(* Logix 5000 project; controller DIMTER vendor 1 type 14 code 77 rev 15.4; software revision 15.01; part 4 of 4 *)
(* tags used below, declared in another part *)
   BufferReady : TIMER;
   CurrentShift : DINT;   // Shift Currently Operating
   F : BOOL[2016];   // Flags
   FLASHER : TIMER;   // Lamp Flasher
   Oneshots : BOOL[128];
   RecordFault : BOOL;
   RecordPieceSaw1 : BOOL;   // Record Piece Count For Shift Total
   RecordPieceSaw2 : BOOL;   // Record Piece Count For Shift Total
   Saw1FailureDelay : TIMER;
   Saw2FailureDelay : TIMER;
   T : TIMER[100];   // Timers
   A120 : ALIAS FOR Local:4:O.Data.0;   // O:4.0/0 A12.0 Buffer Selection1
   A121 : ALIAS FOR Local:4:O.Data.1;   // O:4.0/1 A12/1 Buffer Selection 2
   A122 : ALIAS FOR Local:4:O.Data.2;   // O:4.0/2 A12.2 Reset Failure
   A130 : ALIAS FOR Local:4:O.Data.8;   // O:4.0/8 A13.0 Failure Conveyor
   A131 : ALIAS FOR Local:4:O.Data.9;   // O:4.0/9 A13.1 Failure Saw 1
   A132 : ALIAS FOR Local:4:O.Data.10;   // O:4.0/10 A13.2 Failure Saw 2
   A133 : ALIAS FOR Local:4:O.Data.11;   // O:4.0/11 A13.3 Defect Measuring Computer
   A134 : ALIAS FOR Local:4:O.Data.12;   // O:4.0/12 A13.4 Safety Barrier Transfer Station
   A137 : ALIAS FOR Local:4:O.Data.15;   // O:4.0/15 A137 Safety Barrier Transfer Station
   Delay : TIMER[30];   // Delay Timers
   E00 : ALIAS FOR Local:1:I.Data.0;   // I:1.0/0 E0.0 Control Power On
   E01 : ALIAS FOR Local:1:I.Data.1;   // I:1.0/1 E0.1 Saw Hood 1 Closed
   E02 : ALIAS FOR Local:1:I.Data.2;   // I:1.0/2 E0.2 Saw Motor 1 On
   E03 : ALIAS FOR Local:1:I.Data.3;   // I:1.0/3 E0.3 Release - Feed Saw 1
   E04 : ALIAS FOR Local:1:I.Data.4;   // I:1.0/4 E0.4 Failure Saw 1
   E05 : ALIAS FOR Local:1:I.Data.5;   // I:1.0/5 E0.5 Failure Chain Ejector
   E06 : ALIAS FOR Local:1:I.Data.6;   // I:1.0/6 E0.6 Failure Conveyor in Front of Saw 1
   E07 : ALIAS FOR Local:1:I.Data.7;   // I:1.0/7 E0.7 Failure Conveyor in Front of Saw 2
   E10 : ALIAS FOR Local:1:I.Data.8;   // I:1.0/8 E1.0 Failure Weinig Conveyor
   E106 : ALIAS FOR Local:3:I.Data.22;   // I:3.1/6 E10.6 Cross Belt 1 Cyclewise Continuous Running
   E11 : ALIAS FOR Local:1:I.Data.9;   // I:1.0/9 E1.1 Saw Hood 2 Closed
   E111 : ALIAS FOR Local:3:I.Data.25;   // I:3.1/9 E11.1 Cross Belt 2 Cyclewise Continuous Running
   E12 : ALIAS FOR Local:1:I.Data.10;   // I:1.0/10 E1.2 Saw Motor 2 On
   E13 : ALIAS FOR Local:1:I.Data.11;   // I:1.0/11 E1.3 Release - Feed Saw 2
   E14 : ALIAS FOR Local:1:I.Data.12;   // I:1.0/12 E1.4 Failure Saw 2
   E15 : ALIAS FOR Local:1:I.Data.13;   // I:1.0/13 E1.5 Data Ready At Saw
   E17 : ALIAS FOR Local:1:I.Data.15;   // I:1.0/15 E1.7 Defect Measuring Computer
   E20 : ALIAS FOR Local:1:I.Data.16;   // I:1.1/0 E2.0 Protection Hood Measuring System
   E22 : ALIAS FOR Local:1:I.Data.18;   // I:1.1/2 E2.2 Frequency Converter Rollcase in Front of Saw 1 Ready For Operation
   E23 : ALIAS FOR Local:1:I.Data.19;   // I:1.1/3 E2.3 Frequency Converter Rollcase in Front of Saw 2 Ready For Operation
   E24 : ALIAS FOR Local:1:I.Data.20;   // I:1.1/4 E2.4 Emergency Shutdown Internal
   E26 : ALIAS FOR Local:1:I.Data.22;   // I:1.1/6 E2.6 Safety Barrier at Transfer Station Closed
   E27 : ALIAS FOR Local:1:I.Data.23;   // I:1.1/7 E2.7 Reset Safety Barrier at Transfer Station
   E33 : ALIAS FOR Local:1:I.Data.27;   // I:1/1/11 E3.3 PE Behind Measurement Station
   E43 : ALIAS FOR Local:2:I.Data.3;   // I:2.0/3 E4.3 Infeed Saw 1 On
   E44 : ALIAS FOR Local:2:I.Data.4;   // I:2.0/4 E4.4 Waste Conveyor Belt On
   E47 : ALIAS FOR Local:2:I.Data.7;   // I:2.0/7 E4.7 Lamp Test
   E53 : ALIAS FOR Local:2:I.Data.11;   // I:2.0/11 E5.3 Infeed Saw 2 On
   E54 : ALIAS FOR Local:2:I.Data.12;   // I:2.0/12 E5.4 Measuring Station On
   Faults : BOOL[224];   // Fault Array
   HMI_IntWords : INT[200];   // Integer Words to HMI
   IntsFromHMI : INT[100];   // Integers From HMI
   RealTimeClock : DINT[10];
   Status : BOOL[224];   // Status Array
(* MainProgram, continued *)

ROUTINE ShiftControl   (* ladder *)
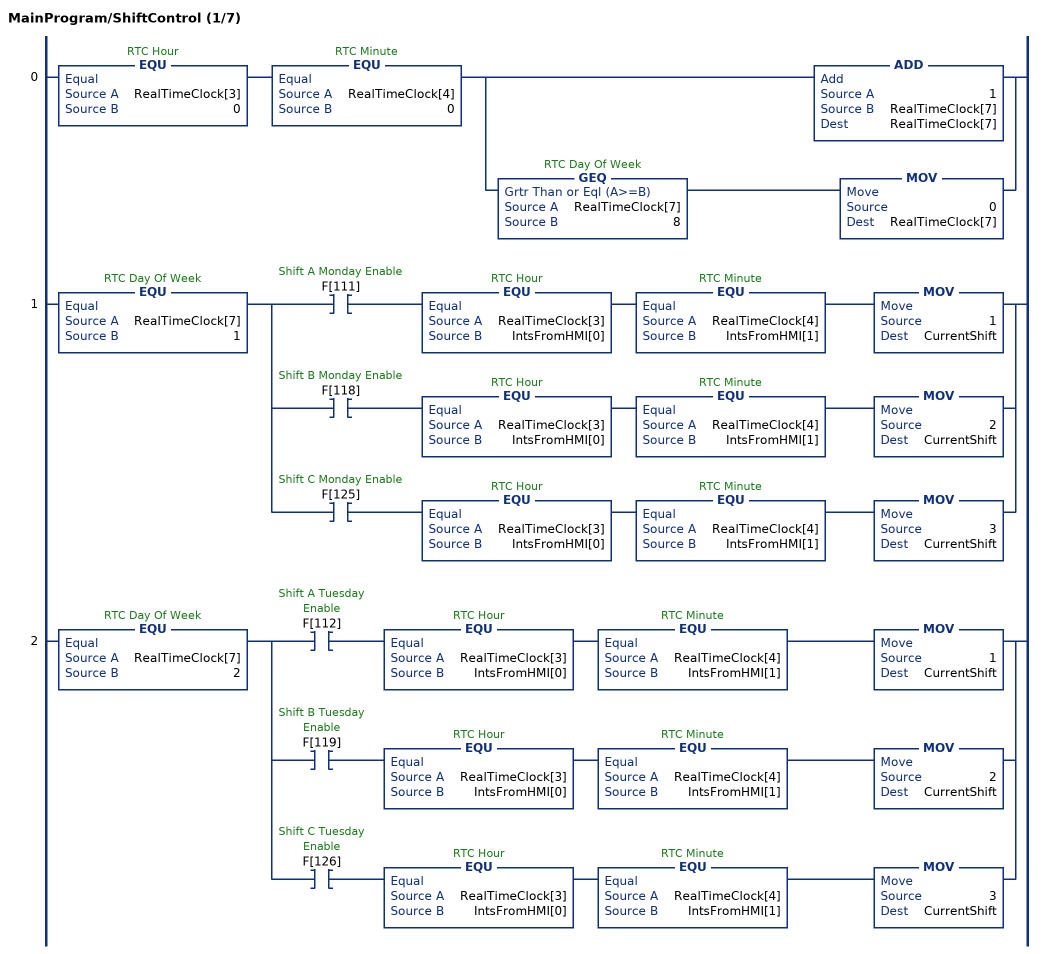
   0: EQU(RealTimeClock[3],0)EQU(RealTimeClock[4],0)[ADD(1,RealTimeClock[7],RealTimeClock[7]) ,GEQ(RealTimeClock[7],8) MOV(0,RealTimeClock[7]) ];
   1: EQU(RealTimeClock[7],1)[XIC(F[111]) EQU(RealTimeClock[3],IntsFromHMI[0]) EQU(RealTimeClock[4],IntsFromHMI[1]) MOV(1,CurrentShift) ,XIC(F[118]) EQU(RealTimeClock[3],IntsFromHMI[0]) EQU(RealTimeClock[4],IntsFromHMI[1]) MOV(2,CurrentShift) ,XIC(F[125]) EQU(RealTimeClock[3],IntsFromHMI[0]) EQU(RealTimeClock[4],IntsFromHMI[1]) MOV(3,CurrentShift) ];
   2: EQU(RealTimeClock[7],2)[XIC(F[112]) EQU(RealTimeClock[3],IntsFromHMI[0]) EQU(RealTimeClock[4],IntsFromHMI[1]) MOV(1,CurrentShift) ,XIC(F[119]) EQU(RealTimeClock[3],IntsFromHMI[0]) EQU(RealTimeClock[4],IntsFromHMI[1]) MOV(2,CurrentShift) ,XIC(F[126]) EQU(RealTimeClock[3],IntsFromHMI[0]) EQU(RealTimeClock[4],IntsFromHMI[1]) MOV(3,CurrentShift) ];
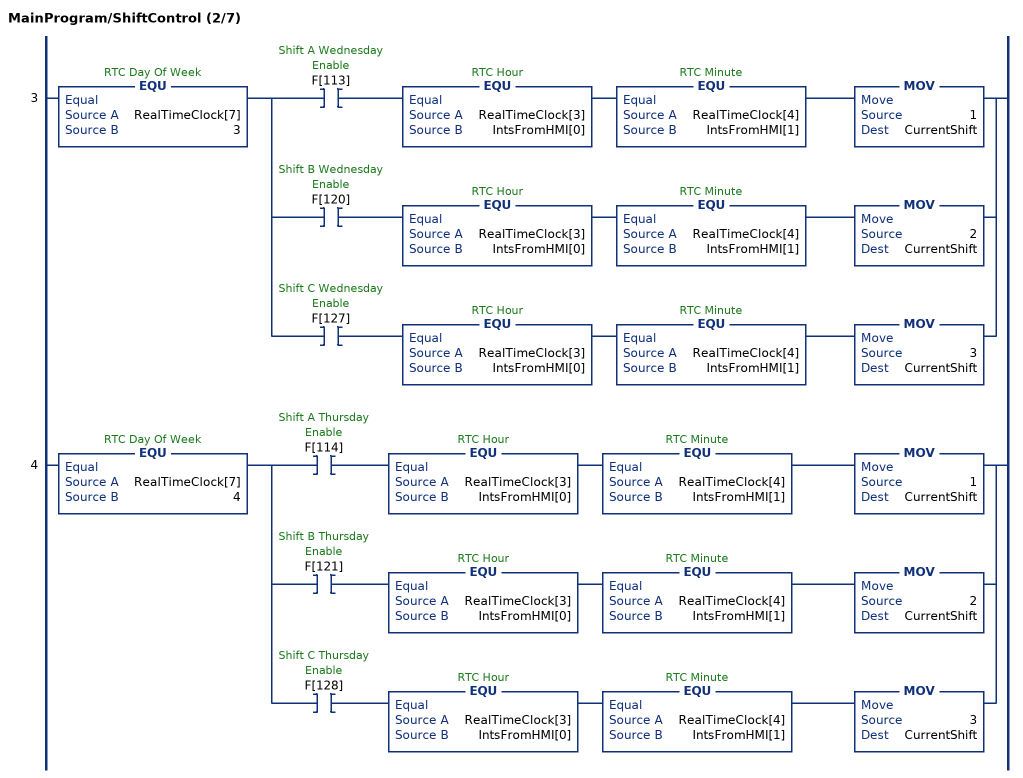
   3: EQU(RealTimeClock[7],3)[XIC(F[113]) EQU(RealTimeClock[3],IntsFromHMI[0]) EQU(RealTimeClock[4],IntsFromHMI[1]) MOV(1,CurrentShift) ,XIC(F[120]) EQU(RealTimeClock[3],IntsFromHMI[0]) EQU(RealTimeClock[4],IntsFromHMI[1]) MOV(2,CurrentShift) ,XIC(F[127]) EQU(RealTimeClock[3],IntsFromHMI[0]) EQU(RealTimeClock[4],IntsFromHMI[1]) MOV(3,CurrentShift) ];
   4: EQU(RealTimeClock[7],4)[XIC(F[114]) EQU(RealTimeClock[3],IntsFromHMI[0]) EQU(RealTimeClock[4],IntsFromHMI[1]) MOV(1,CurrentShift) ,XIC(F[121]) EQU(RealTimeClock[3],IntsFromHMI[0]) EQU(RealTimeClock[4],IntsFromHMI[1]) MOV(2,CurrentShift) ,XIC(F[128]) EQU(RealTimeClock[3],IntsFromHMI[0]) EQU(RealTimeClock[4],IntsFromHMI[1]) MOV(3,CurrentShift) ];
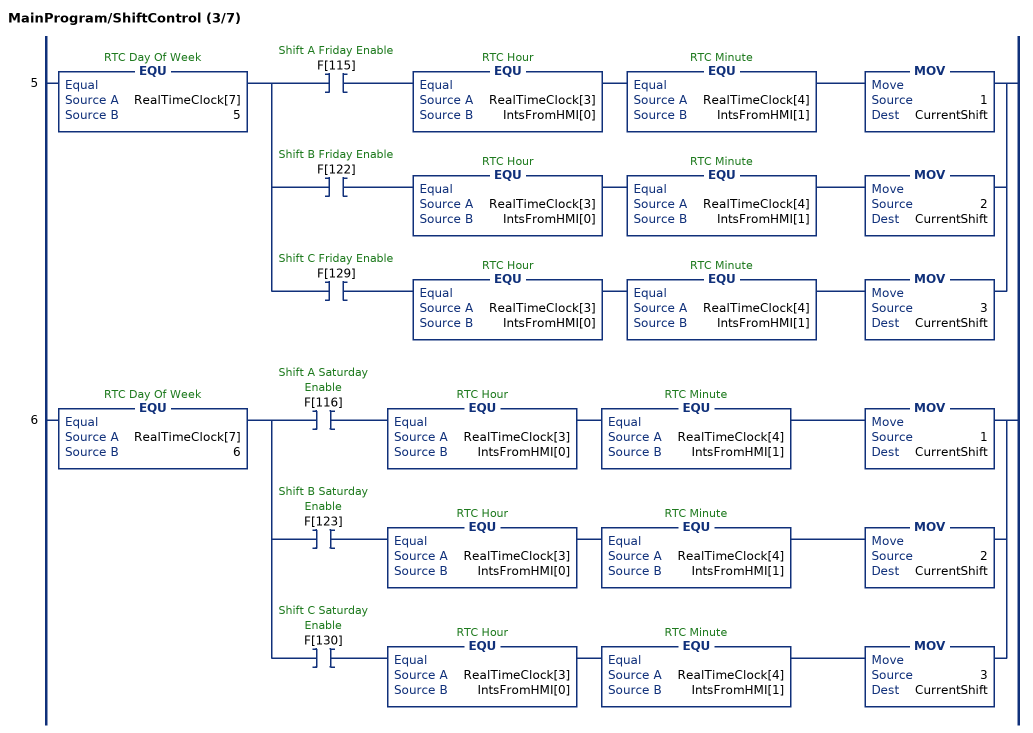
   5: EQU(RealTimeClock[7],5)[XIC(F[115]) EQU(RealTimeClock[3],IntsFromHMI[0]) EQU(RealTimeClock[4],IntsFromHMI[1]) MOV(1,CurrentShift) ,XIC(F[122]) EQU(RealTimeClock[3],IntsFromHMI[0]) EQU(RealTimeClock[4],IntsFromHMI[1]) MOV(2,CurrentShift) ,XIC(F[129]) EQU(RealTimeClock[3],IntsFromHMI[0]) EQU(RealTimeClock[4],IntsFromHMI[1]) MOV(3,CurrentShift) ];
   6: EQU(RealTimeClock[7],6)[XIC(F[116]) EQU(RealTimeClock[3],IntsFromHMI[0]) EQU(RealTimeClock[4],IntsFromHMI[1]) MOV(1,CurrentShift) ,XIC(F[123]) EQU(RealTimeClock[3],IntsFromHMI[0]) EQU(RealTimeClock[4],IntsFromHMI[1]) MOV(2,CurrentShift) ,XIC(F[130]) EQU(RealTimeClock[3],IntsFromHMI[0]) EQU(RealTimeClock[4],IntsFromHMI[1]) MOV(3,CurrentShift) ];
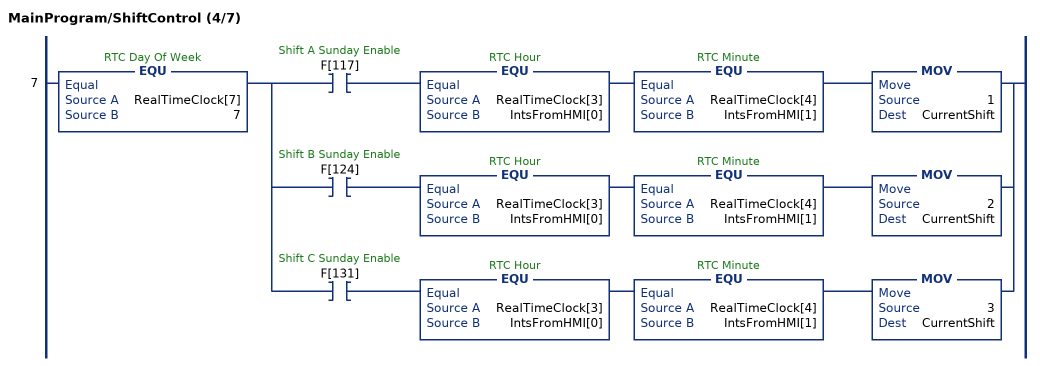
   7: EQU(RealTimeClock[7],7)[XIC(F[117]) EQU(RealTimeClock[3],IntsFromHMI[0]) EQU(RealTimeClock[4],IntsFromHMI[1]) MOV(1,CurrentShift) ,XIC(F[124]) EQU(RealTimeClock[3],IntsFromHMI[0]) EQU(RealTimeClock[4],IntsFromHMI[1]) MOV(2,CurrentShift) ,XIC(F[131]) EQU(RealTimeClock[3],IntsFromHMI[0]) EQU(RealTimeClock[4],IntsFromHMI[1]) MOV(3,CurrentShift) ];
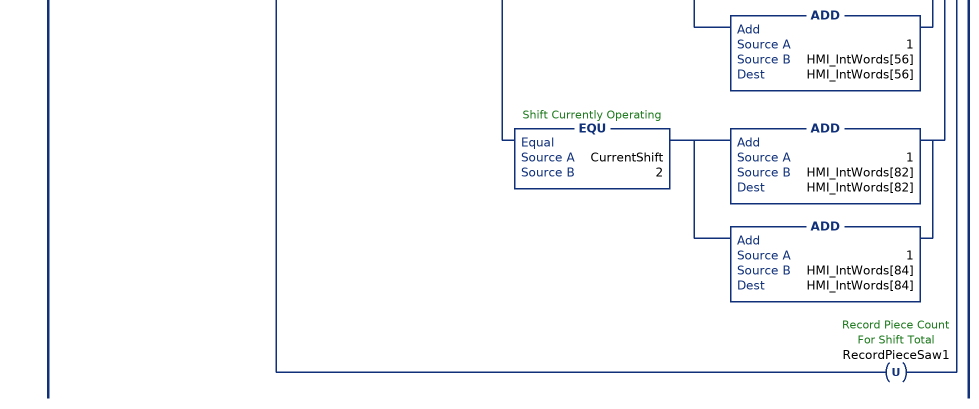
   8: XIC(RecordPieceSaw1)ONS(Oneshots[24])[EQU(RealTimeClock[7],1) [EQU(CurrentShift,1) [ADD(1,HMI_IntWords[2],HMI_IntWords[2]) ,ADD(1,HMI_IntWords[4],HMI_IntWords[4]) ] ,EQU(CurrentShift,2) [ADD(1,HMI_IntWords[30],HMI_IntWords[30]) ,ADD(1,HMI_IntWords[32],HMI_IntWords[32]) ] ,EQU(CurrentShift,2) [ADD(1,HMI_IntWords[58],HMI_IntWords[58]) ,ADD(1,HMI_IntWords[60],HMI_IntWords[60]) ] ] ,EQU(RealTimeClock[7],2) [EQU(CurrentShift,1) [ADD(1,HMI_IntWords[6],HMI_IntWords[6]) ,ADD(1,HMI_IntWords[8],HMI_IntWords[8]) ] ,EQU(CurrentShift,2) [ADD(1,HMI_IntWords[34],HMI_IntWords[34]) ,ADD(1,HMI_IntWords[36],HMI_IntWords[36]) ] ,EQU(CurrentShift,2) [ADD(1,HMI_IntWords[62],HMI_IntWords[62]) ,ADD(1,HMI_IntWords[64],HMI_IntWords[64]) ] ] ,EQU(RealTimeClock[7],3) [EQU(CurrentShift,1) [ADD(1,HMI_IntWords[10],HMI_IntWords[10]) ,ADD(1,HMI_IntWords[12],HMI_IntWords[12]) ] ,EQU(CurrentShift,2) [ADD(1,HMI_IntWords[38],HMI_IntWords[38]) ,ADD(1,HMI_IntWords[40],HMI_IntWords[40]) ] ,EQU(CurrentShift,2) [ADD(1,HMI_IntWords[66],HMI_IntWords[66]) ,ADD(1,HMI_IntWords[68],HMI_IntWords[68]) ] ] ,EQU(RealTimeClock[7],4) [EQU(CurrentShift,1) [ADD(1,HMI_IntWords[14],HMI_IntWords[14]) ,ADD(1,HMI_IntWords[16],HMI_IntWords[16]) ] ,EQU(CurrentShift,2) [ADD(1,HMI_IntWords[42],HMI_IntWords[42]) ,ADD(1,HMI_IntWords[44],HMI_IntWords[44]) ] ,EQU(CurrentShift,2) [ADD(1,HMI_IntWords[70],HMI_IntWords[70]) ,ADD(1,HMI_IntWords[72],HMI_IntWords[72]) ] ] ,EQU(RealTimeClock[7],5) [EQU(CurrentShift,1) [ADD(1,HMI_IntWords[18],HMI_IntWords[18]) ,ADD(1,HMI_IntWords[20],HMI_IntWords[20]) ] ,EQU(CurrentShift,2) [ADD(1,HMI_IntWords[46],HMI_IntWords[46]) ,ADD(1,HMI_IntWords[48],HMI_IntWords[48]) ] ,EQU(CurrentShift,2) [ADD(1,HMI_IntWords[74],HMI_IntWords[74]) ,ADD(1,HMI_IntWords[76],HMI_IntWords[76]) ] ] ,EQU(RealTimeClock[7],6) [EQU(CurrentShift,1) [ADD(1,HMI_IntWords[22],HMI_IntWords[22]) ,ADD(1,HMI_IntWords[24],HMI_IntWords[24]) ] ,EQU(CurrentShift,2) [ADD(1,HMI_IntWords[50],HMI_IntWords[50]) ,ADD(1,HMI_IntWords[52],HMI_IntWords[52]) ] ,EQU(CurrentShift,2) [ADD(1,HMI_IntWords[78],HMI_IntWords[78]) ,ADD(1,HMI_IntWords[80],HMI_IntWords[80]) ] ] ,EQU(RealTimeClock[7],7) [EQU(CurrentShift,1) [ADD(1,HMI_IntWords[26],HMI_IntWords[26]) ,ADD(1,HMI_IntWords[28],HMI_IntWords[28]) ] ,EQU(CurrentShift,2) [ADD(1,HMI_IntWords[54],HMI_IntWords[54]) ,ADD(1,HMI_IntWords[56],HMI_IntWords[56]) ] ,EQU(CurrentShift,2) [ADD(1,HMI_IntWords[82],HMI_IntWords[82]) ,ADD(1,HMI_IntWords[84],HMI_IntWords[84]) ] ] ,OTU(RecordPieceSaw1) ];
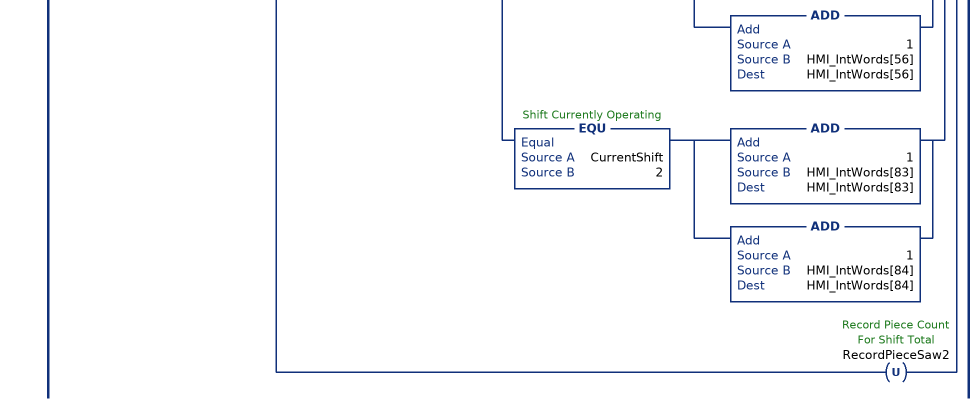
   9: XIC(RecordPieceSaw2)ONS(Oneshots[25])[EQU(RealTimeClock[7],1) [EQU(CurrentShift,1) [ADD(1,HMI_IntWords[3],HMI_IntWords[3]) ,ADD(1,HMI_IntWords[4],HMI_IntWords[4]) ] ,EQU(CurrentShift,2) [ADD(1,HMI_IntWords[31],HMI_IntWords[31]) ,ADD(1,HMI_IntWords[32],HMI_IntWords[32]) ] ,EQU(CurrentShift,2) [ADD(1,HMI_IntWords[59],HMI_IntWords[59]) ,ADD(1,HMI_IntWords[60],HMI_IntWords[60]) ] ] ,EQU(RealTimeClock[7],2) [EQU(CurrentShift,1) [ADD(1,HMI_IntWords[7],HMI_IntWords[7]) ,ADD(1,HMI_IntWords[8],HMI_IntWords[8]) ] ,EQU(CurrentShift,2) [ADD(1,HMI_IntWords[35],HMI_IntWords[35]) ,ADD(1,HMI_IntWords[36],HMI_IntWords[36]) ] ,EQU(CurrentShift,2) [ADD(1,HMI_IntWords[63],HMI_IntWords[63]) ,ADD(1,HMI_IntWords[64],HMI_IntWords[64]) ] ] ,EQU(RealTimeClock[7],3) [EQU(CurrentShift,1) [ADD(1,HMI_IntWords[11],HMI_IntWords[11]) ,ADD(1,HMI_IntWords[12],HMI_IntWords[12]) ] ,EQU(CurrentShift,2) [ADD(1,HMI_IntWords[39],HMI_IntWords[39]) ,ADD(1,HMI_IntWords[40],HMI_IntWords[40]) ] ,EQU(CurrentShift,2) [ADD(1,HMI_IntWords[67],HMI_IntWords[67]) ,ADD(1,HMI_IntWords[68],HMI_IntWords[68]) ] ] ,EQU(RealTimeClock[7],4) [EQU(CurrentShift,1) [ADD(1,HMI_IntWords[15],HMI_IntWords[15]) ,ADD(1,HMI_IntWords[16],HMI_IntWords[16]) ] ,EQU(CurrentShift,2) [ADD(1,HMI_IntWords[43],HMI_IntWords[43]) ,ADD(1,HMI_IntWords[44],HMI_IntWords[44]) ] ,EQU(CurrentShift,2) [ADD(1,HMI_IntWords[71],HMI_IntWords[71]) ,ADD(1,HMI_IntWords[72],HMI_IntWords[72]) ] ] ,EQU(RealTimeClock[7],5) [EQU(CurrentShift,1) [ADD(1,HMI_IntWords[19],HMI_IntWords[19]) ,ADD(1,HMI_IntWords[20],HMI_IntWords[20]) ] ,EQU(CurrentShift,2) [ADD(1,HMI_IntWords[47],HMI_IntWords[47]) ,ADD(1,HMI_IntWords[48],HMI_IntWords[48]) ] ,EQU(CurrentShift,2) [ADD(1,HMI_IntWords[75],HMI_IntWords[75]) ,ADD(1,HMI_IntWords[76],HMI_IntWords[76]) ] ] ,EQU(RealTimeClock[7],6) [EQU(CurrentShift,1) [ADD(1,HMI_IntWords[23],HMI_IntWords[23]) ,ADD(1,HMI_IntWords[24],HMI_IntWords[24]) ] ,EQU(CurrentShift,2) [ADD(1,HMI_IntWords[51],HMI_IntWords[51]) ,ADD(1,HMI_IntWords[52],HMI_IntWords[52]) ] ,EQU(CurrentShift,2) [ADD(1,HMI_IntWords[79],HMI_IntWords[79]) ,ADD(1,HMI_IntWords[80],HMI_IntWords[80]) ] ] ,EQU(RealTimeClock[7],7) [EQU(CurrentShift,1) [ADD(1,HMI_IntWords[27],HMI_IntWords[27]) ,ADD(1,HMI_IntWords[28],HMI_IntWords[28]) ] ,EQU(CurrentShift,2) [ADD(1,HMI_IntWords[55],HMI_IntWords[55]) ,ADD(1,HMI_IntWords[56],HMI_IntWords[56]) ] ,EQU(CurrentShift,2) [ADD(1,HMI_IntWords[83],HMI_IntWords[83]) ,ADD(1,HMI_IntWords[84],HMI_IntWords[84]) ] ] ,OTU(RecordPieceSaw2) ];
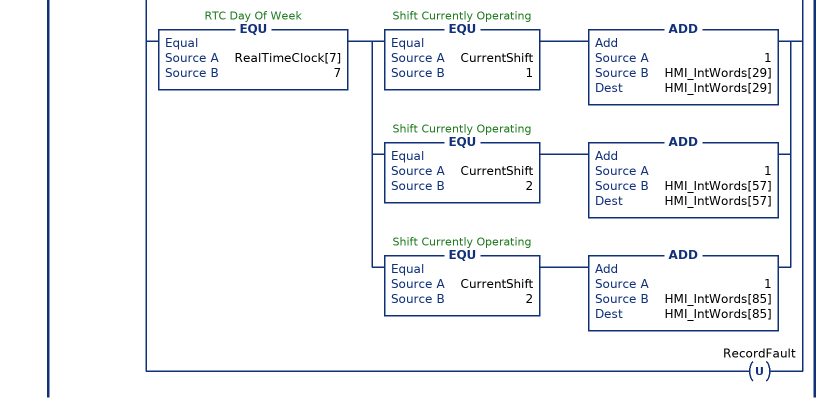
   10: XIC(RecordFault)[EQU(RealTimeClock[7],1) [EQU(CurrentShift,1) ADD(1,HMI_IntWords[5],HMI_IntWords[5]) ,EQU(CurrentShift,2) ADD(1,HMI_IntWords[33],HMI_IntWords[33]) ,EQU(CurrentShift,2) ADD(1,HMI_IntWords[61],HMI_IntWords[61]) ] ,EQU(RealTimeClock[7],2) [EQU(CurrentShift,1) ADD(1,HMI_IntWords[9],HMI_IntWords[9]) ,EQU(CurrentShift,2) ADD(1,HMI_IntWords[37],HMI_IntWords[37]) ,EQU(CurrentShift,2) ADD(1,HMI_IntWords[65],HMI_IntWords[65]) ] ,EQU(RealTimeClock[7],3) [EQU(CurrentShift,1) ADD(1,HMI_IntWords[13],HMI_IntWords[13]) ,EQU(CurrentShift,2) ADD(1,HMI_IntWords[41],HMI_IntWords[41]) ,EQU(CurrentShift,2) ADD(1,HMI_IntWords[69],HMI_IntWords[69]) ] ,EQU(RealTimeClock[7],4) [EQU(CurrentShift,1) ADD(1,HMI_IntWords[17],HMI_IntWords[17]) ,EQU(CurrentShift,2) ADD(1,HMI_IntWords[45],HMI_IntWords[45]) ,EQU(CurrentShift,2) ADD(1,HMI_IntWords[73],HMI_IntWords[73]) ] ,EQU(RealTimeClock[7],5) [EQU(CurrentShift,1) ADD(1,HMI_IntWords[21],HMI_IntWords[21]) ,EQU(CurrentShift,2) ADD(1,HMI_IntWords[49],HMI_IntWords[49]) ,EQU(CurrentShift,2) ADD(1,HMI_IntWords[77],HMI_IntWords[77]) ] ,EQU(RealTimeClock[7],6) [EQU(CurrentShift,1) ADD(1,HMI_IntWords[25],HMI_IntWords[25]) ,EQU(CurrentShift,2) ADD(1,HMI_IntWords[53],HMI_IntWords[53]) ,EQU(CurrentShift,2) ADD(1,HMI_IntWords[81],HMI_IntWords[81]) ] ,EQU(RealTimeClock[7],7) [EQU(CurrentShift,1) ADD(1,HMI_IntWords[29],HMI_IntWords[29]) ,EQU(CurrentShift,2) ADD(1,HMI_IntWords[57],HMI_IntWords[57]) ,EQU(CurrentShift,2) ADD(1,HMI_IntWords[85],HMI_IntWords[85]) ] ,OTU(RecordFault) ];
END_ROUTINE

ROUTINE Status   (* ladder *)
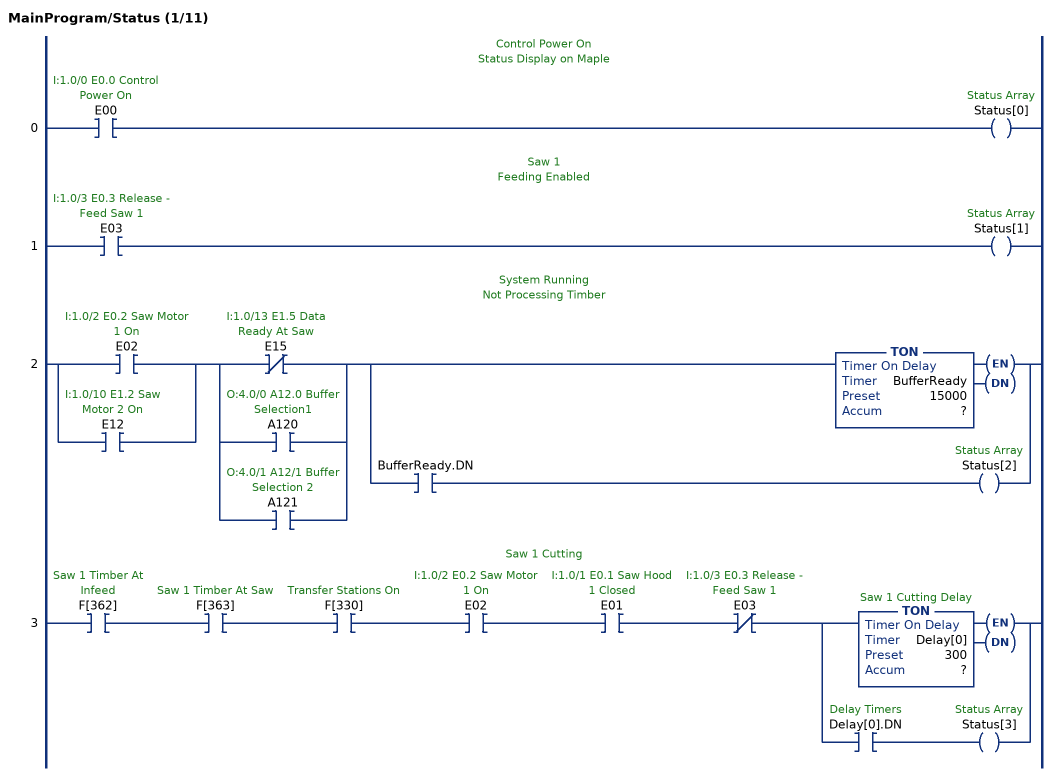
   // Control Power On
   // Status Display on Maple
   0: XIC(E00)OTE(Status[0]);
   // Saw 1
   // Feeding Enabled
   1: XIC(E03)OTE(Status[1]);
   // System Running
   // Not Processing Timber
   2: [XIC(E02) ,XIC(E12) ][XIO(E15) ,XIC(A120) ,XIC(A121) ][TON(BufferReady,?,?) ,XIC(BufferReady.DN) OTE(Status[2]) ];
   // Saw 1 Cutting
   3: XIC(F[362])XIC(F[363])XIC(F[330])XIC(E02)XIC(E01)XIO(E03)[TON(Delay[0],?,?) ,XIC(Delay[0].DN) OTE(Status[3]) ];
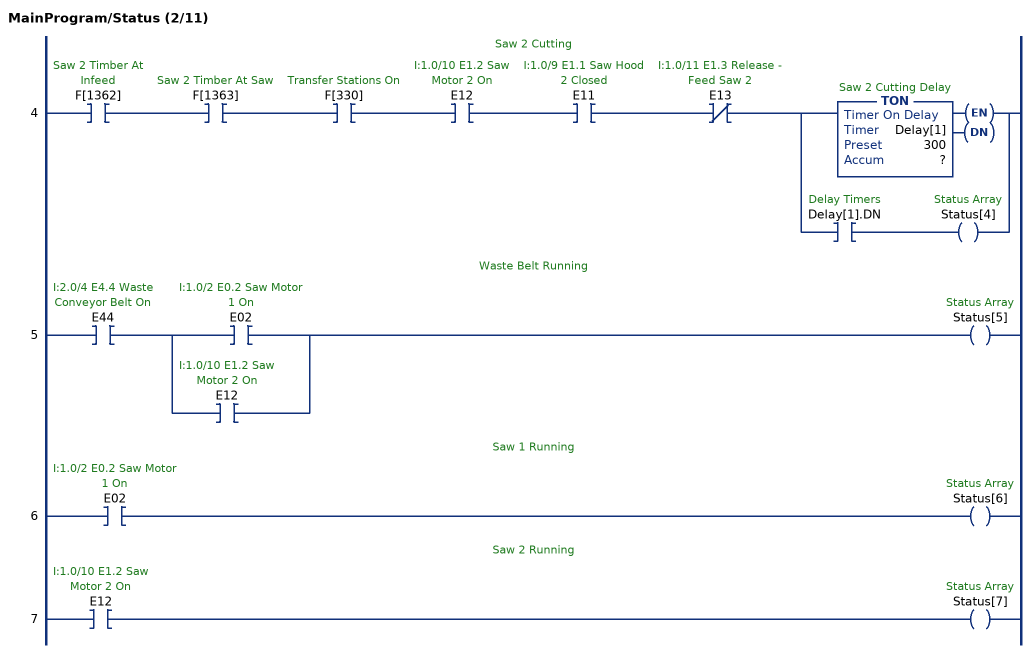
   // Saw 2 Cutting
   4: XIC(F[1362])XIC(F[1363])XIC(F[330])XIC(E12)XIC(E11)XIO(E13)[TON(Delay[1],?,?) ,XIC(Delay[1].DN) OTE(Status[4]) ];
   // Waste Belt Running
   5: XIC(E44)[XIC(E02) ,XIC(E12) ]OTE(Status[5]);
   // Saw 1 Running
   6: XIC(E02)OTE(Status[6]);
   // Saw 2 Running
   7: XIC(E12)OTE(Status[7]);
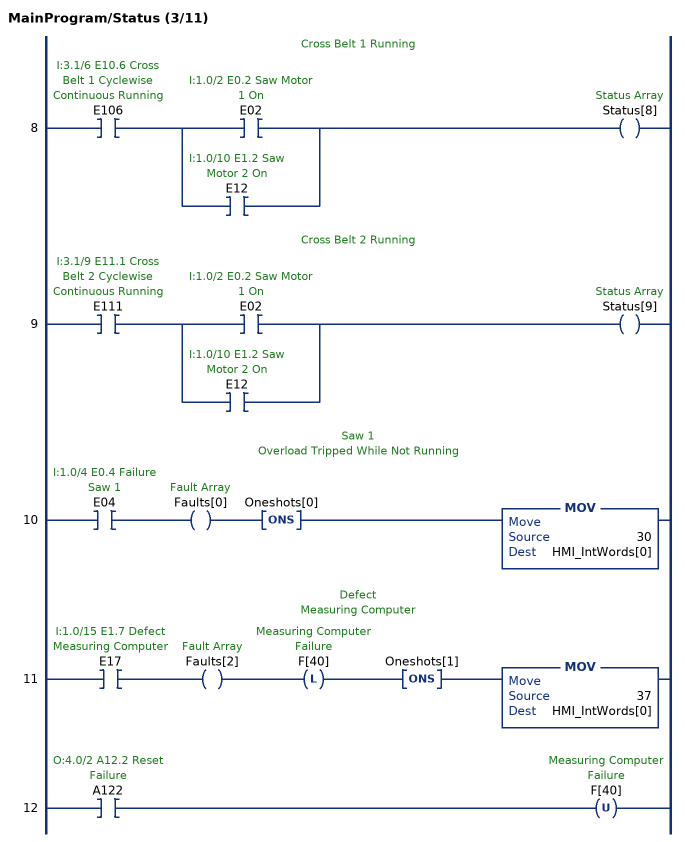
   // Cross Belt 1 Running
   8: XIC(E106)[XIC(E02) ,XIC(E12) ]OTE(Status[8]);
   // Cross Belt 2 Running
   9: XIC(E111)[XIC(E02) ,XIC(E12) ]OTE(Status[9]);
   // Saw 1
   // Overload Tripped While Not Running
   10: XIC(E04)OTE(Faults[0])ONS(Oneshots[0])MOV(30,HMI_IntWords[0]);
   // Defect
   // Measuring Computer
   11: XIC(E17)OTE(Faults[2])OTL(F[40])ONS(Oneshots[1])MOV(37,HMI_IntWords[0]);
   12: XIC(A122)OTU(F[40]);
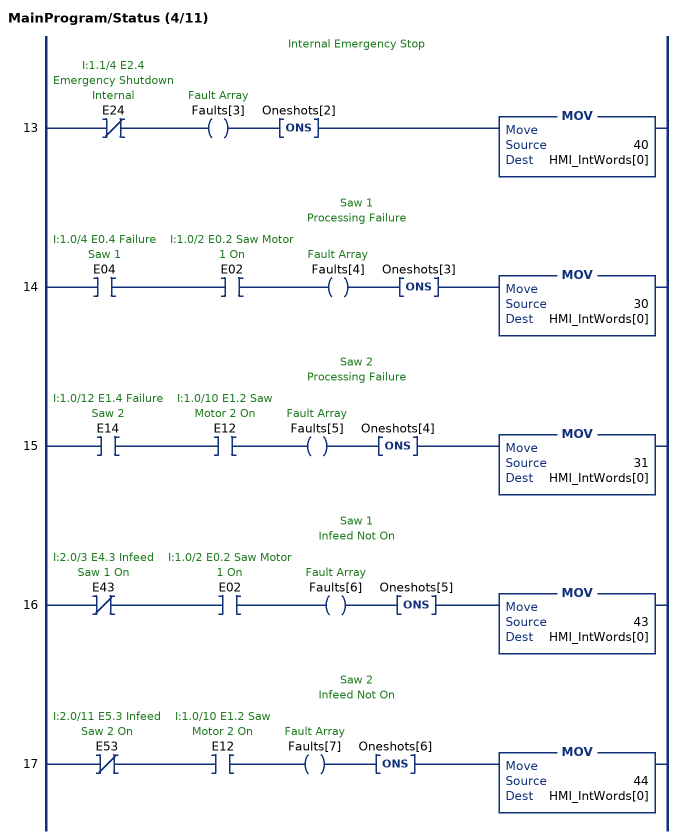
   // Internal Emergency Stop
   13: XIO(E24)OTE(Faults[3])ONS(Oneshots[2])MOV(40,HMI_IntWords[0]);
   // Saw 1
   // Processing Failure
   14: XIC(E04)XIC(E02)OTE(Faults[4])ONS(Oneshots[3])MOV(30,HMI_IntWords[0]);
   // Saw 2
   // Processing Failure
   15: XIC(E14)XIC(E12)OTE(Faults[5])ONS(Oneshots[4])MOV(31,HMI_IntWords[0]);
   // Saw 1
   // Infeed Not On
   16: XIO(E43)XIC(E02)OTE(Faults[6])ONS(Oneshots[5])MOV(43,HMI_IntWords[0]);
   // Saw 2
   // Infeed Not On
   17: XIO(E53)XIC(E12)OTE(Faults[7])ONS(Oneshots[6])MOV(44,HMI_IntWords[0]);
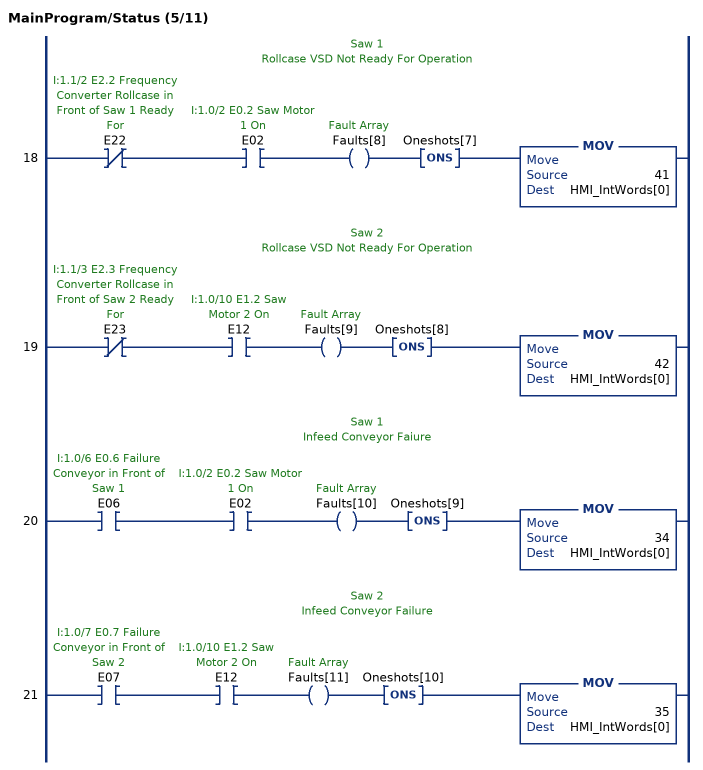
   // Saw 1
   // Rollcase VSD Not Ready For Operation
   18: XIO(E22)XIC(E02)OTE(Faults[8])ONS(Oneshots[7])MOV(41,HMI_IntWords[0]);
   // Saw 2
   // Rollcase VSD Not Ready For Operation
   19: XIO(E23)XIC(E12)OTE(Faults[9])ONS(Oneshots[8])MOV(42,HMI_IntWords[0]);
   // Saw 1
   // Infeed Conveyor Faiure
   20: XIC(E06)XIC(E02)OTE(Faults[10])ONS(Oneshots[9])MOV(34,HMI_IntWords[0]);
   // Saw 2
   // Infeed Conveyor Failure
   21: XIC(E07)XIC(E12)OTE(Faults[11])ONS(Oneshots[10])MOV(35,HMI_IntWords[0]);
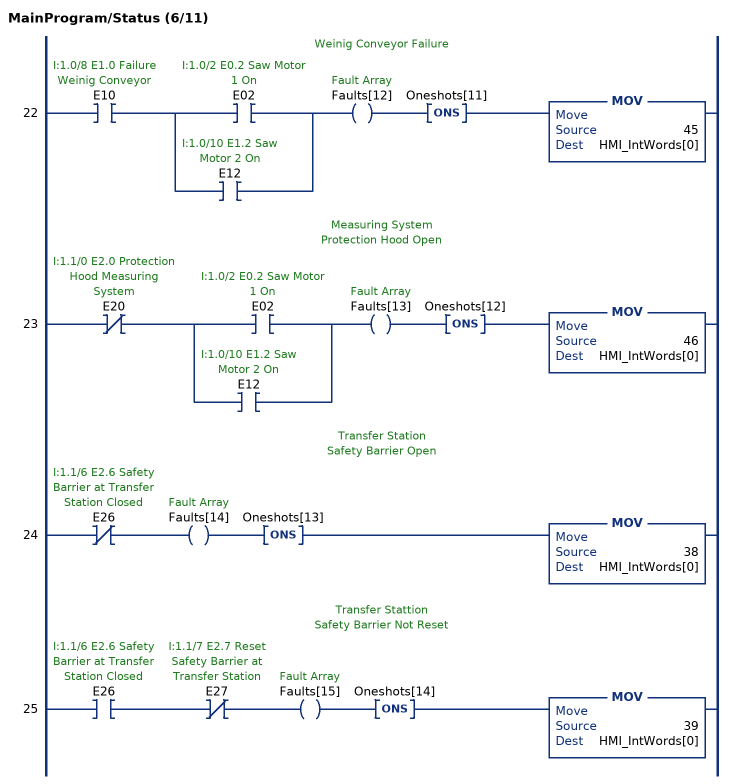
   // Weinig Conveyor Failure
   22: XIC(E10)[XIC(E02) ,XIC(E12) ]OTE(Faults[12])ONS(Oneshots[11])MOV(45,HMI_IntWords[0]);
   // Measuring System
   // Protection Hood Open
   23: XIO(E20)[XIC(E02) ,XIC(E12) ]OTE(Faults[13])ONS(Oneshots[12])MOV(46,HMI_IntWords[0]);
   // Transfer Station
   // Safety Barrier Open
   24: XIO(E26)OTE(Faults[14])ONS(Oneshots[13])MOV(38,HMI_IntWords[0]);
   // Transfer Stattion
   // Safety Barrier Not Reset
   25: XIC(E26)XIO(E27)OTE(Faults[15])ONS(Oneshots[14])MOV(39,HMI_IntWords[0]);
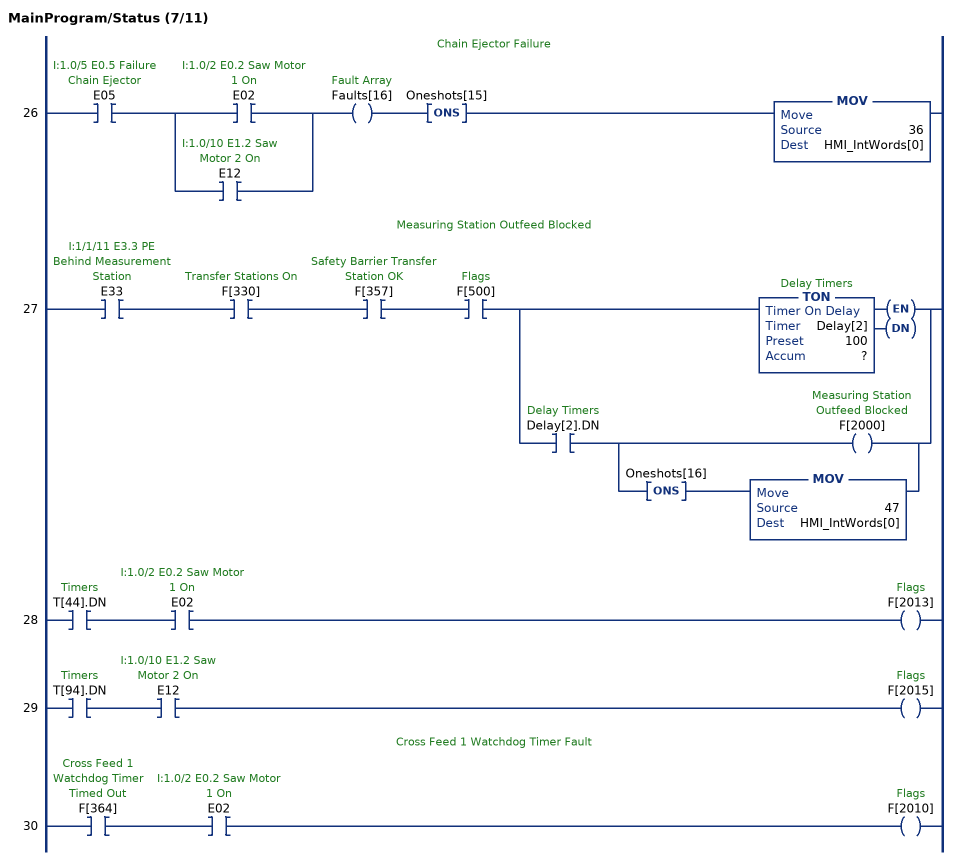
   // Chain Ejector Failure
   26: XIC(E05)[XIC(E02) ,XIC(E12) ]OTE(Faults[16])ONS(Oneshots[15])MOV(36,HMI_IntWords[0]);
   // Measuring Station Outfeed Blocked
   27: XIC(E33)XIC(F[330])XIC(F[357])XIC(F[500])[TON(Delay[2],?,?) ,XIC(Delay[2].DN) [OTE(F[2000]) ,ONS(Oneshots[16]) MOV(47,HMI_IntWords[0]) ] ];
   28: XIC(T[44].DN)XIC(E02)OTE(F[2013]);
   29: XIC(T[94].DN)XIC(E12)OTE(F[2015]);
   // Cross Feed 1 Watchdog Timer Fault
   30: XIC(F[364])XIC(E02)OTE(F[2010]);
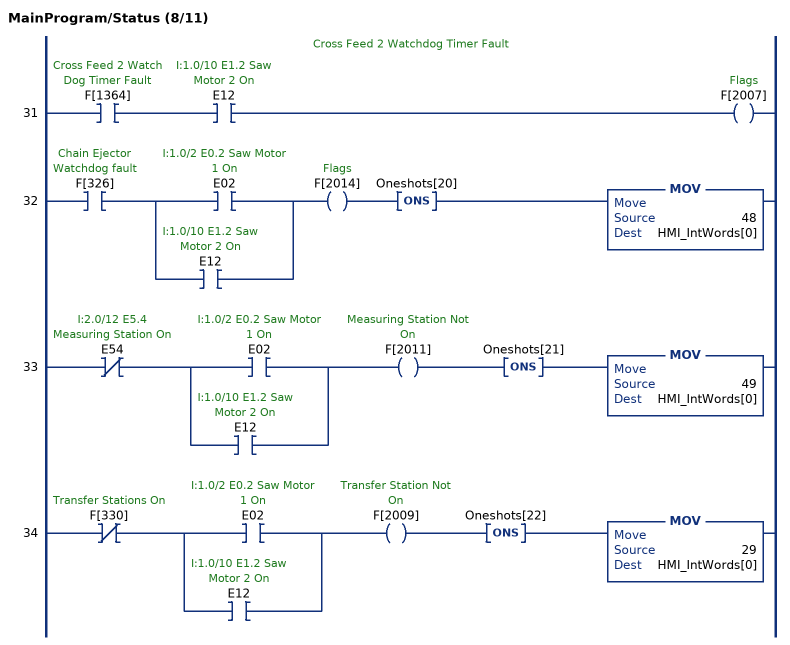
   // Cross Feed 2 Watchdog Timer Fault
   31: XIC(F[1364])XIC(E12)OTE(F[2007]);
   32: XIC(F[326])[XIC(E02) ,XIC(E12) ]OTE(F[2014])ONS(Oneshots[20])MOV(48,HMI_IntWords[0]);
   33: XIO(E54)[XIC(E02) ,XIC(E12) ]OTE(F[2011])ONS(Oneshots[21])MOV(49,HMI_IntWords[0]);
   34: XIO(F[330])[XIC(E02) ,XIC(E12) ]OTE(F[2009])ONS(Oneshots[22])MOV(29,HMI_IntWords[0]);
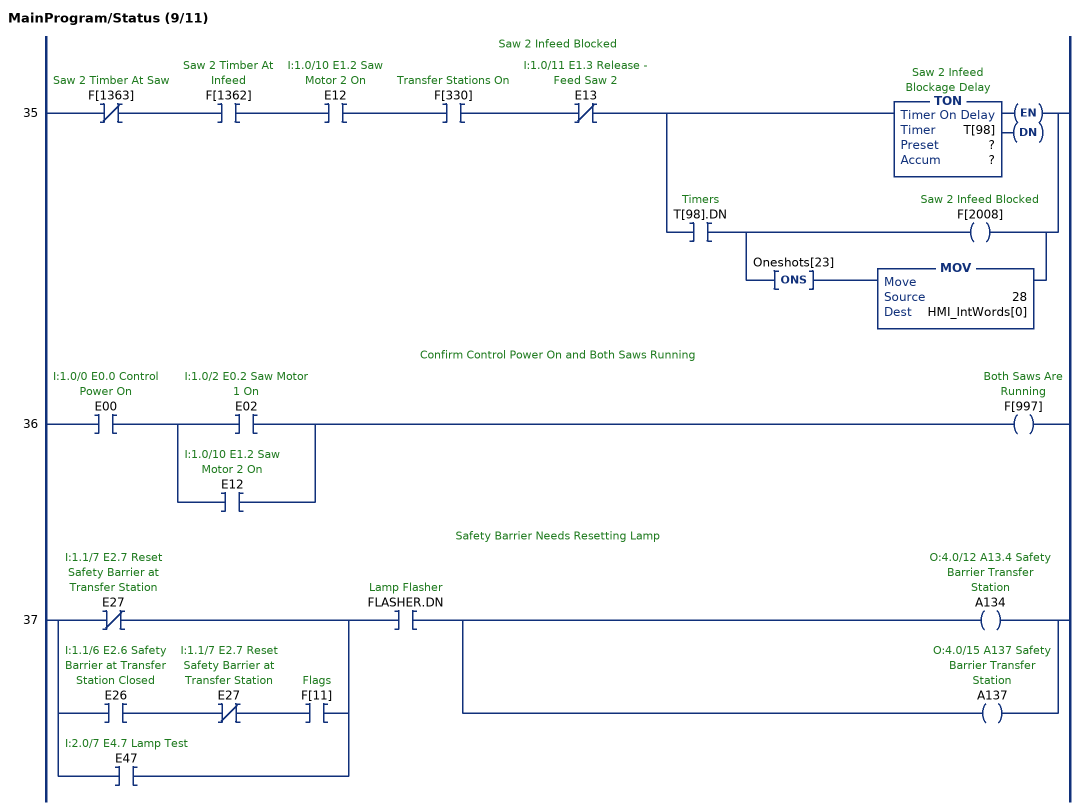
   // Saw 2 Infeed Blocked
   35: XIO(F[1363])XIC(F[1362])XIC(E12)XIC(F[330])XIO(E13)[TON(T[98],?,?) ,XIC(T[98].DN) [OTE(F[2008]) ,ONS(Oneshots[23]) MOV(28,HMI_IntWords[0]) ] ];
   // Confirm Control Power On and Both Saws Running
   36: XIC(E00)[XIC(E02) ,XIC(E12) ]OTE(F[997]);
   // Safety Barrier Needs Resetting Lamp
   37: [XIO(E27) ,[XIC(E26) XIO(E27) XIC(F[11]) ,XIC(E47) ] ]XIC(FLASHER.DN)[OTE(A134) ,OTE(A137) ];
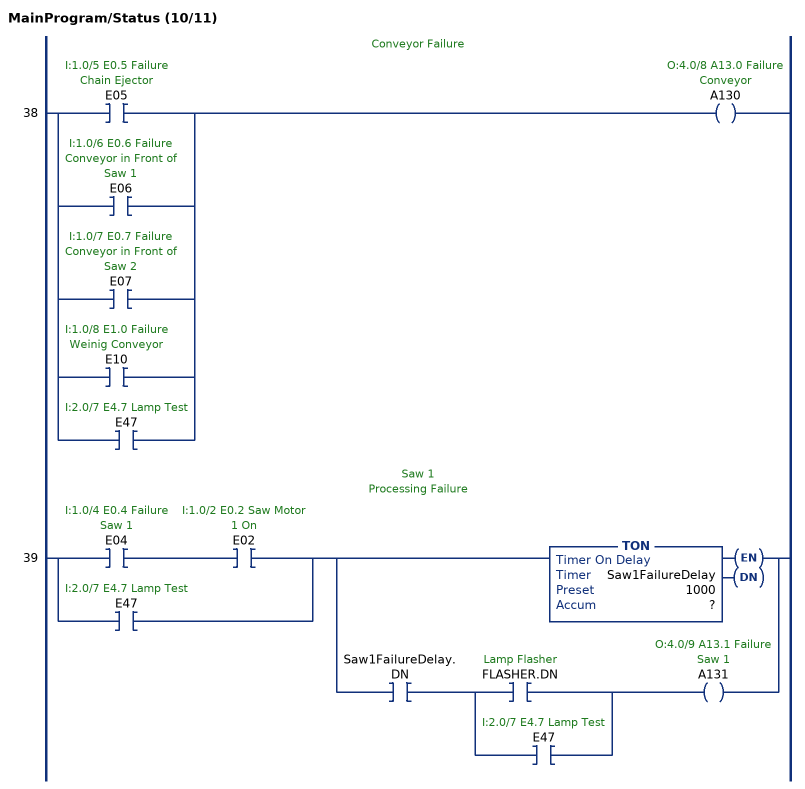
   // Conveyor Failure
   38: [XIC(E05) ,XIC(E06) ,XIC(E07) ,XIC(E10) ,XIC(E47) ]OTE(A130);
   // Saw 1
   // Processing Failure
   39: [XIC(E04) XIC(E02) ,XIC(E47) ][TON(Saw1FailureDelay,?,?) ,XIC(Saw1FailureDelay.DN) [XIC(FLASHER.DN) ,XIC(E47) ] OTE(A131) ];
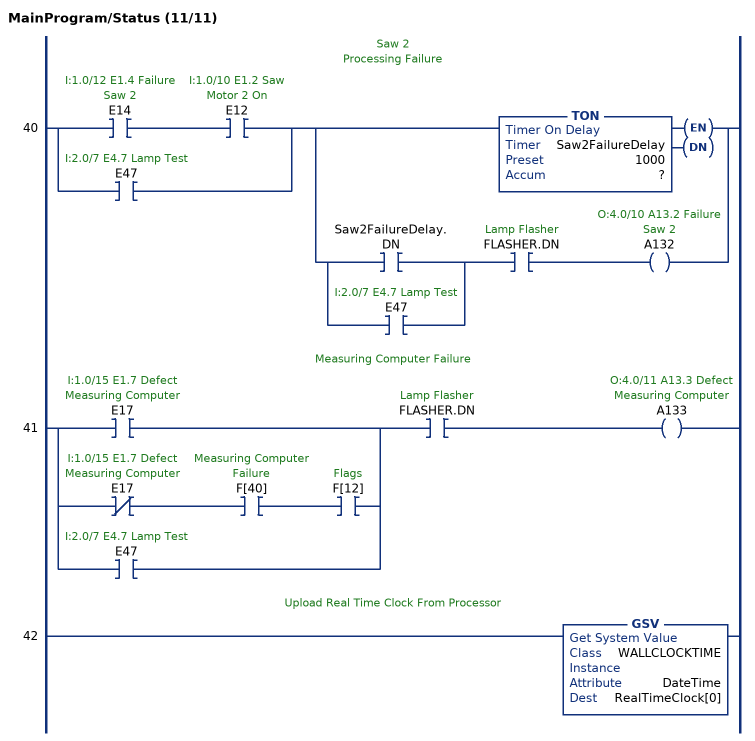
   // Saw 2
   // Processing Failure
   40: [XIC(E14) XIC(E12) ,XIC(E47) ][TON(Saw2FailureDelay,?,?) ,[XIC(Saw2FailureDelay.DN) ,XIC(E47) ] XIC(FLASHER.DN) OTE(A132) ];
   // Measuring Computer Failure
   41: [XIC(E17) ,XIO(E17) XIC(F[40]) XIC(F[12]) ,XIC(E47) ]XIC(FLASHER.DN)OTE(A133);
   // Upload Real Time Clock From Processor
   42: GSV(WALLCLOCKTIME,,DateTime,RealTimeClock[0]);
END_ROUTINE
END_PROGRAM
